{attribute 'Tc2GvlVarNames'}
{attribute 'strict'}
TYPE e_StatoCentratura :
(
	CENTRATURA_DISABILITATA		:= 0, 
	CENTRATURA_DA_ESEGUIRE	:= 1, 
	CENTRATURA_ESEGUITA 		:= 2
);
END_TYPE

(* stored: Version 1.1.0.1, ProductVersion 3.1.4024.11
   DUT e_StatoCentratura: Id {3cbff908-b72e-4a0b-9e92-6f1b1d5d81b4} *)
